FUNCTION_BLOCK FB_SolSolPiston_2Pos
VAR_INPUT
    (* Automatic Commands from PLC sequence logic. Wired to FALSE in MAIN until FB_Auto exists. *)
    bAutoCmdExtend    : BOOL;
    bAutoCmdRetract   : BOOL;

    (* Physical Feedback (Proximity Switches) *)
    bSwitchExtended   : BOOL;
    bSwitchRetracted  : BOOL;
END_VAR

VAR_IN_OUT
    (* HMI contract — mode, manual + simulate inputs, latched + sensor status *)
    stHmi             : ST_HmiPiston;
END_VAR

VAR_OUTPUT
    (* Physical Outputs to Solenoids *)
    bOutSolenoidExtend  : BOOL;
    bOutSolenoidRetract : BOOL;
END_VAR

VAR
    (* Internal Target States *)
    bTargetExtend     : BOOL;
    bTargetRetract    : BOOL;

    (* HMI Manual-Button Edge Detection *)
    fbTrigManExtend   : R_TRIG;
    fbTrigManRetract  : R_TRIG;

    (* Effective sensor states = real OR HMI simulate. Recomputed every cycle in Section 0a. *)
    bSwitchExtended_eff  : BOOL;
    bSwitchRetracted_eff : BOOL;
END_VAR

(* ==========================================
   0a. EFFECTIVE SENSOR INPUTS (real OR HMI simulate)
   ========================================== *)
bSwitchExtended_eff  := bSwitchExtended  OR stHmi.bSimulateExtended;
bSwitchRetracted_eff := bSwitchRetracted OR stHmi.bSimulateRetracted;

(* ==========================================
   0. HMI MANUAL BUTTON LATCHING (Radio-Button Behavior)
   ========================================== *)
fbTrigManExtend(CLK := stHmi.bManCmdExtend);
fbTrigManRetract(CLK := stHmi.bManCmdRetract);

// Independent IFs (not ELSIF): if multiple edges fire in the same cycle, the last one wins (Retract > Extend).
IF fbTrigManExtend.Q  THEN stHmi.bSelectedExtend := TRUE;  stHmi.bSelectedRetract := FALSE; END_IF;
IF fbTrigManRetract.Q THEN stHmi.bSelectedExtend := FALSE; stHmi.bSelectedRetract := TRUE;  END_IF;

IF stHmi.eMode = E_ControlMode.Automatic THEN
    stHmi.bSelectedExtend := FALSE; stHmi.bSelectedRetract := FALSE;
END_IF;

(* ==========================================
   1. MODE SELECTION & COMMAND MAPPING
   ========================================== *)
IF stHmi.eMode = E_ControlMode.Automatic THEN
    bTargetExtend  := bAutoCmdExtend;
    bTargetRetract := bAutoCmdRetract;

ELSIF stHmi.eMode = E_ControlMode.Manual THEN
    bTargetExtend  := stHmi.bSelectedExtend;
    bTargetRetract := stHmi.bSelectedRetract;

ELSE
    // Safe default: undefined mode → no targets
    bTargetExtend  := FALSE;
    bTargetRetract := FALSE;
END_IF;

(* ==========================================
   1b. TARGET-REACHED RESET — clear bSelected* once the piston arrives
   ========================================== *)
IF stHmi.bSelectedExtend  AND bSwitchExtended_eff  THEN stHmi.bSelectedExtend  := FALSE; END_IF;
IF stHmi.bSelectedRetract AND bSwitchRetracted_eff THEN stHmi.bSelectedRetract := FALSE; END_IF;

(* ==========================================
   2. SOLENOID CONTROL
   ========================================== *)
// CASE 1: Move to EXTENDED position
IF bTargetExtend AND NOT bSwitchExtended_eff THEN
    bOutSolenoidExtend  := TRUE;
    bOutSolenoidRetract := FALSE;

// CASE 2: Move to RETRACTED position
ELSIF bTargetRetract AND NOT bSwitchRetracted_eff THEN
    bOutSolenoidRetract := TRUE;
    bOutSolenoidExtend  := FALSE;

// CASE 3: Target reached or no active target → stop both coils
ELSE
    bOutSolenoidExtend  := FALSE;
    bOutSolenoidRetract := FALSE;
END_IF;

(* ==========================================
   3. HMI STATUS FEEDBACK
   ========================================== *)
stHmi.bIsExtended        := bSwitchExtended_eff;
stHmi.bIsRetracted       := bSwitchRetracted_eff;
stHmi.bIsMoving          := bOutSolenoidExtend OR bOutSolenoidRetract;
stHmi.bOutSolenoidExtend  := bOutSolenoidExtend;
stHmi.bOutSolenoidRetract := bOutSolenoidRetract;

END_FUNCTION_BLOCK

(* stored: Version 1.1.0.1, ProductVersion 3.1.4026.18
   POU FB_SolSolPiston_2Pos: Id {1cc505ad-12b3-4ad6-b3e6-2111bf6da3c3}, SpecialFunc None *)
